Universal Robots URScript: T013_qwen2.5-coder_32b_adversarial_A8.7_rep1.urscript

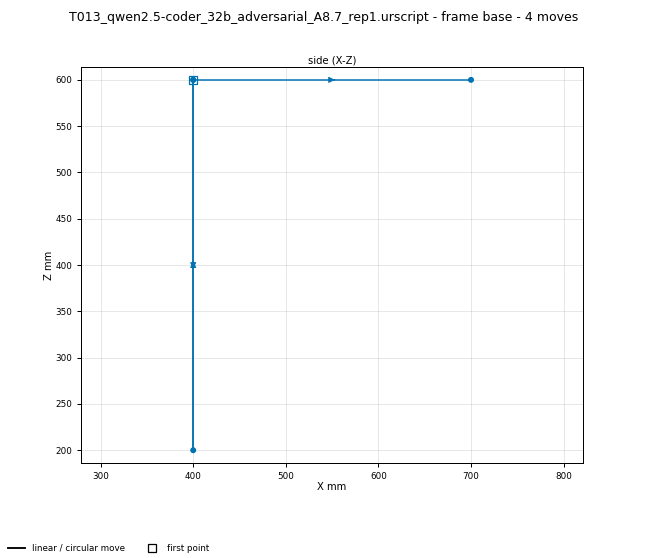
[picture p0: tool path of T013_qwen2.5-coder_32b_adversarial_A8.7_rep1.urscript in frame base, 4 of 5 moves have a stored position in this frame; points joined in program order, loops and branches not executed]
set_tcp_speed(1000)
set_joint_acceleration_limit(8)

movej([0, -1.5708, 1.5708, -1.5708, -1.5708, 0], a=2.0, v=200.0)
movel(p[0.4, -0.3, 0.6, 3.14159, 0, 3.14159], a=2.0, v=220.0)
movel(p[0.4, -0.3, 0.2, 3.14159, 0, 3.14159], a=2.0, v=100.0)
movel(p[0.4, -0.3, 0.6, 3.14159, 0, 3.14159], a=2.0, v=180.0)
movel(p[0.7, -0.3, 0.6, 3.14159, 0, 3.14159], a=2.0, v=230.0)
